# EPICS autosave request: elveFlowESmobileApp/Db/elveFlow_settings.req
$(P)$(R)Pres1
$(P)$(R)P1TweakVal
